TYPE DS_BrensonEnclosure :
STRUCT
	DSBrensonGenerator : ARRAY [1..iUSGeneratorQty] OF DS_BrensonGenerator;
END_STRUCT
END_TYPE

(* stored: Version 1.1.0.1, ProductVersion 3.1.4024.12
   DUT DS_BrensonEnclosure: Id {da40e28e-4b39-4b09-9bd2-0692aed1f458} *)
